PROGRAM knoppen
VAR
	bmagneet	    AT %Q* : BOOL;
	bpomp1			AT %Q* : BOOL;
	bpomp2			AT %Q* : BOOL;
END_VAR

END_PROGRAM

(* stored: Version 1.1.0.1, ProductVersion 3.1.4024.2
   POU knoppen: Id {6c143f2d-6165-4a19-8917-831738003274}, SpecialFunc None *)
